FUNCTION_BLOCK RecordableStation001_Components EXTENDS TcoCore.TcoObject
VAR	
	{attribute addProperty Name "Horizontal cyclinder A1"}
	_horizontal : fbPiston(THIS^);
	{attribute addProperty Name "Vertical cyclinder A2"}
	_vertical : fbPiston(THIS^);
	{attribute addProperty Name "Gripper A3"}
	_gripper : fbPiston(THIS^);		
	
END_VAR

VAR
	_simTimerValue : UINT := 500;
	_simTimer : Tc2_Standard.TON;
END_VAR

_vertical();
_horizontal();
_gripper();

PROPERTY Gripper : IPistonGripper
GET
Gripper := _gripper;
END_GET
END_PROPERTY

PROPERTY Horizontal : IPistonHorizontal
GET
Horizontal := _horizontal;
END_GET
END_PROPERTY

METHOD Service
VAR_INPUT
END_VAR
THIS^._gripper.Service();
THIS^._horizontal.Service();
THIS^._vertical.Service();
END_METHOD

PROPERTY Vertical : IPistonVertical
GET
Vertical := _vertical;
END_GET
END_PROPERTY

END_FUNCTION_BLOCK

(* stored: Version 1.1.0.1
   POU RecordableStation001_Components: Id {c710b5bd-0ebb-05bd-1fb5-392d36f4c0e1}, SpecialFunc None
   Property Gripper: Id {369d32ce-c2b1-0e4b-2ff8-5a385e18cf05}
   Get Get: Id {8d48bc6e-90ef-0fa0-1d6e-0247cc4a19bc}
   Property Horizontal: Id {999a82c9-1ecc-0b7a-287e-45dbd9009925}
   Get Get: Id {a2931c7a-4a78-00b9-1dbb-b9d1d205e39d}
   Method Service: Id {855df606-77d4-055d-1b08-c87c84912d93}
   Property Vertical: Id {5216e68a-5d7e-04e5-2c97-2cf00c76fdd4}
   Get Get: Id {846eb78d-cb93-053a-1f89-c73b7a348e46} *)
